// TwinCAT 3 PLC project MR1L0_MR2L0_PLC
// ProgramVersion: 3.1.4022.7
// libraries:
//   Tc2_ControllerToolbox, * (Beckhoff Automation GmbH)
//   Tc2_MC2, * (Beckhoff Automation GmbH)
//   Tc2_SerialCom, * (Beckhoff Automation GmbH)
//   Tc2_Standard, * (Beckhoff Automation GmbH)
//   Tc2_System, * (Beckhoff Automation GmbH)
//   Tc2_Utilities, * (Beckhoff Automation GmbH)
//   Tc3_Module, * (Beckhoff Automation GmbH)
//   VisuDialogs, * (System)
//   LCLS General,0.0.0,SLAC
//   lcls-twincat-motion,1.1.0,SLAC
//   lcls-twincat-optics,0.0.0,SLAC
// project tree:
//   / GlobalTextList.TcGTLO, PiezoDriver.TcTTO (not stored), PlcTask.TcTTO, SerialIO.TcTTO, Visualization Manager.TcVMO (not stored)
//   GVLs/ GVL_COM_Buffers.TcGVL, GVL_M1L0.TcGVL, GVL_M1L0_Constants.TcGVL, GVL_M2L0.TcGVL, GVL_M2L0_Constants.TcGVL, GVL_SerialIO.TcGVL
//   POUs/ Main.TcPOU
//   POUs/Serial Comm/ PiezoSerial.TcPOU, P_Serial_Com.TcPOU
// real-time tasks:
//   TASK PlcTask: cycle T#10ms, priority 20, ADS port 350
//   TASK PiezoDriver: cycle T#1ms, priority 3, ADS port 351
//   TASK SerialIO: cycle T#2ms, priority 1, ADS port 352
// motion (NC):
//   TASK NC-Task 1 SAF: cycle T#2ms, priority 4, ADS port 501
//   TASK NC-Task 1 SVB: cycle T#10ms, priority 8, ADS port 511
//   AXIS M1L0-Yup (id 1)
//     General: UnitName=um
//     Dynamic: Acceleration=200, Deceleration=200, DelayTime=0.008
//     Velo: Maximum=200
//     OtherSettings: AllowMotionCmdToSlave=true
//     encoder EncType=29
//       EncPara: ScaleFactorNumerator=0.001, MaxCount=#xffffffff, ReferenceSystem=1
//         SoftEndMinControl: Enable=true, Range=3133.7
//         SoftEndMaxControl: Enable=true, Range=27004.8
//         Inc: RefSoftSyncMask=#x0000ffff
//     drive DrvType=24
//       DrvPara: Inverse=true
//         Analog: VeloReferenz=488.28125, ScaleFactorActTorque=0.1
//         TimeComp: TaskDelayCycles=1
//     controller CtrType=2
//       CtrPara: PriorControlFactor=1
//         PosDiffControl: Range=100
//         PID: PosKp=50, PosExtKp=10, DeadBandPosition=0.3
//         Observer: BandWidth=20
//   AXIS M1L0-Ydwn (id 2)
//     General: UnitName=um
//     Dynamic: Acceleration=200, Deceleration=200, DelayTime=0.008
//     Velo: Maximum=200
//     OtherSettings: AllowMotionCmdToSlave=true
//     encoder EncType=29
//       EncPara: ScaleFactorNumerator=0.001, MaxCount=#xffffffff, ReferenceSystem=1
//         SoftEndMinControl: Enable=true, Range=2244.7
//         SoftEndMaxControl: Enable=true, Range=26310.2
//         Inc: RefSoftSyncMask=#x0000ffff
//     drive DrvType=24
//       DrvPara: Inverse=true
//         Analog: VeloReferenz=488.28125, ScaleFactorActTorque=0.1
//         TimeComp: TaskDelayCycles=1
//     controller CtrType=2
//       CtrPara: PriorControlFactor=1
//         PosDiffControl: Range=100
//         PID: PosKp=50, PosExtKp=10, DeadBandPosition=0.3
//         Observer: BandWidth=20
//   AXIS M1L0-Xup (id 3)
//     General: UnitName=um
//     Dynamic: Acceleration=2000, Deceleration=2000, DelayTime=0.008
//     Velo: Maximum=1000
//     OtherSettings: AllowMotionCmdToSlave=true
//     encoder EncType=29
//       EncPara: ScaleFactorNumerator=0.001, MaxCount=#xffffffff, ReferenceSystem=1
//         SoftEndMinControl: Enable=true, Range=24843
//         SoftEndMaxControl: Enable=true, Range=25581.9
//         Inc: RefSoftSyncMask=#x0000ffff
//     drive DrvType=24
//       Analog: VeloReferenz=1220.703125, ScaleFactorActTorque=0.1
//       TimeComp: TaskDelayCycles=1
//     controller CtrType=2
//       CtrPara: PriorControlFactor=1
//         PosDiffControl: Range=100
//         PID: PosKp=50, PosExtKp=50, DeadBandPosition=0.4
//         Observer: BandWidth=20
//   AXIS M1L0-Xdwn (id 4)
//     General: UnitName=um
//     Dynamic: Acceleration=2000, Deceleration=2000, DelayTime=0.008
//     Velo: Maximum=1000
//     OtherSettings: AllowMotionCmdToSlave=true
//     encoder EncType=29
//       EncPara: ScaleFactorNumerator=0.001, MaxCount=#xffffffff, ReferenceSystem=1
//         SoftEndMinControl: Range=24000
//         SoftEndMaxControl: Enable=true, Range=24518.2
//         Inc: RefSoftSyncMask=#x0000ffff
//     drive DrvType=24
//       DrvPara: Inverse=true
//         Analog: VeloReferenz=1220.703125, ScaleFactorActTorque=0.1
//         TimeComp: TaskDelayCycles=1
//     controller CtrType=2
//       CtrPara: PriorControlFactor=1
//         PosDiffControl: Range=100
//         PID: PosKp=50, PosExtKp=50, DeadBandPosition=0.4
//         Observer: BandWidth=20
//   AXIS M1L0-Pitch (id 5)
//     General: UnitName=urad
//     Dynamic: Acceleration=390, Deceleration=390, DelayTime=0.008
//     Velo: Maximum=150
//     OtherSettings: AllowMotionCmdToSlave=true
//     encoder EncType=29
//       EncPara: ScaleFactorNumerator=0.001949317739, MaxCount=#xffffffff, ReferenceSystem=1
//         SoftEndMinControl: Enable=true, Range=15600
//         SoftEndMaxControl: Enable=true, Range=21600
//         Inc: RefSoftSyncMask=#x0000ffff
//     drive DrvType=24
//       Analog: VeloReferenz=761.4522417, ScaleFactorActTorque=0.1
//       TimeComp: TaskDelayCycles=1
//     controller CtrType=2
//       CtrPara: PriorControlFactor=1
//         PosDiffControl: Range=150
//         PID: PosExtKp=1, DeadBandPosition=0.25
//         Observer: BandWidth=20
//   AXIS M1L0-Bender (id 6)
//     General: UnitName=um
//     Dynamic: Acceleration=150, Deceleration=150, DelayTime=0.008
//     Velo: Maximum=150
//     OtherSettings: AllowMotionCmdToSlave=true
//     encoder EncType=29
//       EncPara: ScaleFactorNumerator=0.001, MaxCount=#xffffffff, ReferenceSystem=1
//         SoftEndMinControl: Enable=true, Range=4268900
//         SoftEndMaxControl: Enable=true, Range=4278150
//         Inc: RefSoftSyncMask=#x0000ffff
//     drive DrvType=24
//       DrvPara: Inverse=true
//         Analog: VeloReferenz=195.3125, ScaleFactorActTorque=0.1
//         TimeComp: TaskDelayCycles=1
//     controller CtrType=2
//       CtrPara: PriorControlFactor=1
//         PID: PosKp=10, PosExtKp=0.001, PosExtVelo=0.9, DeadBandPosition=0.1
//         Observer: BandWidth=20
//   AXIS M2L0-Yup (id 7)
//     General: UnitName=um
//     Dynamic: Acceleration=200, Deceleration=200, DelayTime=0.008
//     Velo: Maximum=200
//     OtherSettings: AllowMotionCmdToSlave=true
//     encoder EncType=29
//       EncPara: ScaleFactorNumerator=0.001, MaxCount=#xffffffff, ReferenceSystem=1
//         SoftEndMinControl: Enable=true, Range=2500
//         SoftEndMaxControl: Enable=true, Range=18750
//         Inc: RefSoftSyncMask=#x0000ffff
//     drive DrvType=24
//       DrvPara: Inverse=true
//         Analog: VeloReferenz=488.28125, ScaleFactorActTorque=0.1
//         TimeComp: TaskDelayCycles=1
//     controller CtrType=2
//       CtrPara: PriorControlFactor=1
//         PosDiffControl: Range=100
//         PID: PosKp=20, PosExtKp=5, DeadBandPosition=0.4
//         Observer: BandWidth=20
//   AXIS M2L0-Ydwn (id 8)
//     General: UnitName=um
//     Dynamic: Acceleration=200, Deceleration=200, DelayTime=0.008
//     Velo: Maximum=200
//     OtherSettings: AllowMotionCmdToSlave=true
//     encoder EncType=29
//       EncPara: ScaleFactorNumerator=0.001, MaxCount=#xffffffff, ReferenceSystem=1
//         SoftEndMinControl: Enable=true, Range=5450
//         SoftEndMaxControl: Enable=true, Range=21800
//         Inc: RefSoftSyncMask=#x0000ffff
//     drive DrvType=24
//       DrvPara: Inverse=true
//         Analog: VeloReferenz=488.28125, ScaleFactorActTorque=0.1
//         TimeComp: TaskDelayCycles=1
//     controller CtrType=2
//       CtrPara: PriorControlFactor=1
//         PosDiffControl: Range=100
//         PID: PosKp=20, PosExtKp=5, DeadBandPosition=0.4
//         Observer: BandWidth=20
//   AXIS M2L0-Xup (id 9)
//     General: UnitName=um
//     Dynamic: Acceleration=2000, Deceleration=2000, DelayTime=0.008
//     Velo: Maximum=1000
//     OtherSettings: AllowMotionCmdToSlave=true
//     encoder EncType=29
//       EncPara: ScaleFactorNumerator=0.001, MaxCount=#xffffffff, ReferenceSystem=1
//         SoftEndMinControl: Enable=true, Range=24300
//         SoftEndMaxControl: Enable=true, Range=26200
//         Inc: RefSoftSyncMask=#x0000ffff
//     drive DrvType=24
//       Analog: VeloReferenz=1220.703125, ScaleFactorActTorque=0.1
//       TimeComp: TaskDelayCycles=1
//     controller CtrType=2
//       CtrPara: PriorControlFactor=1
//         PosDiffControl: Range=100
//         PID: PosKp=10, PosExtKp=1, DeadBandPosition=0.4
//         Observer: BandWidth=20
//   AXIS M2L0-Xdwn (id 10)
//     General: UnitName=um
//     Dynamic: Acceleration=2000, Deceleration=2000, DelayTime=0.008
//     Velo: Maximum=1000
//     OtherSettings: AllowMotionCmdToSlave=true
//     encoder EncType=29
//       EncPara: ScaleFactorNumerator=0.001, MaxCount=#xffffffff, ReferenceSystem=1
//         SoftEndMinControl: Range=23500
//         SoftEndMaxControl: Range=25700
//         Inc: RefSoftSyncMask=#x0000ffff
//     drive DrvType=24
//       DrvPara: Inverse=true
//         Analog: VeloReferenz=1220.703125, ScaleFactorActTorque=0.1
//         TimeComp: TaskDelayCycles=1
//     controller CtrType=2
//       CtrPara: PriorControlFactor=1
//         PosDiffControl: Range=100
//         PID: PosKp=10, PosExtKp=1, DeadBandPosition=0.4
//         Observer: BandWidth=20
//   AXIS M2L0-Pitch (id 11)
//     General: UnitName=urad
//     Dynamic: Acceleration=390, Deceleration=390
//     Velo: Maximum=150
//     OtherSettings: AllowMotionCmdToSlave=true
//     encoder EncType=29
//       EncPara: ScaleFactorNumerator=0.001949317739, MaxCount=#xffffffff, ReferenceSystem=1
//         SoftEndMinControl: Enable=true, Range=16200
//         SoftEndMaxControl: Enable=true, Range=20600
//         Inc: RefSoftSyncMask=#x0000ffff
//     drive DrvType=24
//       Analog: VeloReferenz=761.4522417, ScaleFactorActTorque=0.1
//       TimeComp: TaskDelayCycles=1
//     controller CtrType=2
//       CtrPara: PriorControlFactor=1
//         PosDiffControl: Range=150
//         PID: PosExtKp=1, DeadBandPosition=0.2
//         Observer: BandWidth=20
//   AXIS M2L0-Bender (id 12)
//     General: UnitName=um
//     Dynamic: Acceleration=150, Deceleration=150, DelayTime=0.008
//     Velo: Maximum=150
//     OtherSettings: AllowMotionCmdToSlave=true
//     encoder EncType=29
//       EncPara: ScaleFactorNumerator=0.001, MaxCount=#xffffffff, ReferenceSystem=1
//         SoftEndMinControl: Enable=true, Range=4268977
//         SoftEndMaxControl: Enable=true, Range=4279741
//         Inc: RefSoftSyncMask=#x0000ffff
//     drive DrvType=24
//       DrvPara: Inverse=true
//         Analog: VeloReferenz=195.3125, ScaleFactorActTorque=0.1
//         TimeComp: TaskDelayCycles=1
//     controller CtrType=2
//       CtrPara: PriorControlFactor=1
//         PID: PosKp=10, PosExtKp=0.001, PosExtVelo=0.9, DeadBandPosition=0.1
//         Observer: BandWidth=20
// I/O:
//   DEVICE Device 1 (EtherCAT), AmsNetId 172.21.88.30.2.1
//     Term 1 (EK1200)
// variable links:
//   (this object) <-> Device 1 (EtherCAT)/Term 1 (EK1200)/Term 5 (EK1122)/EK1100_M1L0/EL5042_M1L0_Yupdwn
//     Enc/Inputs/In/nComState @bit 1 <-> WcState/InputToggle
//     Enc/Inputs/In/nComState <-> WcState/WcState
//     Enc/Inputs/In/nDataIn1 <-> FB Inputs Channel 1/Position
//     Enc/Inputs/In/nDataIn1 <-> FB Inputs Channel 2/Position
//     Enc/Inputs/In/nState1 @bit 12 <-> FB Inputs Channel 1/Status/Diag
//     Enc/Inputs/In/nState1 @bit 12 <-> FB Inputs Channel 2/Status/Diag
//     Enc/Inputs/In/nState1 @bit 1 <-> FB Inputs Channel 1/Status/Error
//     Enc/Inputs/In/nState1 @bit 1 <-> FB Inputs Channel 2/Status/Error
//     Enc/Inputs/In/nState1 @bit 14 <-> FB Inputs Channel 1/Status/Input cycle counter
//     Enc/Inputs/In/nState1 @bit 14 <-> FB Inputs Channel 2/Status/Input cycle counter
//     Enc/Inputs/In/nState1 @bit 2 <-> FB Inputs Channel 1/Status/Ready
//     Enc/Inputs/In/nState1 @bit 2 <-> FB Inputs Channel 2/Status/Ready
//     Enc/Inputs/In/nState1 @bit 13 <-> FB Inputs Channel 1/Status/TxPDO State
//     Enc/Inputs/In/nState1 @bit 13 <-> FB Inputs Channel 2/Status/TxPDO State
//     Enc/Inputs/In/nState1 <-> FB Inputs Channel 1/Status/Warning
//     Enc/Inputs/In/nState1 <-> FB Inputs Channel 2/Status/Warning
//   (this object) <-> Device 1 (EtherCAT)/Term 1 (EK1200)/Term 5 (EK1122)/EK1100_M1L0/EL7041-1000_M1L0_Yup
//     Drive/Inputs/In/nState1 @bit 3 <-> STM Status/Status/Error
//     Drive/Inputs/In/nState1 @bit 5 <-> STM Status/Status/Moving negative
//     Drive/Inputs/In/nState1 @bit 4 <-> STM Status/Status/Moving positive
//     Drive/Inputs/In/nState1 @bit 1 <-> STM Status/Status/Ready
//     Drive/Inputs/In/nState1 <-> STM Status/Status/Ready to enable
//     Drive/Inputs/In/nState1 @bit 6 <-> STM Status/Status/Torque reduced
//     Drive/Inputs/In/nState1 @bit 2 <-> STM Status/Status/Warning
//     Drive/Inputs/In/nState2 @bit 3 <-> STM Status/Status/Digital input 1
//     Drive/Inputs/In/nState2 @bit 4 <-> STM Status/Status/Digital input 2
//     Drive/Inputs/In/nState2 @bit 5 <-> STM Status/Status/Sync error
//     Drive/Inputs/In/nState2 @bit 7 <-> STM Status/Status/TxPDO Toggle
//     Drive/Inputs/In/nState4 @bit 1 <-> WcState/InputToggle
//     Drive/Inputs/In/nState4 <-> WcState/WcState
//     Drive/Outputs/Out/nCtrl1 <-> STM Control/Control/Enable
//     Drive/Outputs/Out/nCtrl1 @bit 2 <-> STM Control/Control/Reduce torque
//     Drive/Outputs/Out/nCtrl1 @bit 1 <-> STM Control/Control/Reset
//     Drive/Outputs/Out/nDataOut2[0] <-> STM Velocity/Velocity
//   (this object) <-> Device 1 (EtherCAT)/Term 1 (EK1200)/Term 5 (EK1122)/EK1100_M1L0/EL7041-1000_M1L0_Ydwn
//     Drive/Inputs/In/nState1 @bit 3 <-> STM Status/Status/Error
//     Drive/Inputs/In/nState1 @bit 5 <-> STM Status/Status/Moving negative
//     Drive/Inputs/In/nState1 @bit 4 <-> STM Status/Status/Moving positive
//     Drive/Inputs/In/nState1 @bit 1 <-> STM Status/Status/Ready
//     Drive/Inputs/In/nState1 <-> STM Status/Status/Ready to enable
//     Drive/Inputs/In/nState1 @bit 6 <-> STM Status/Status/Torque reduced
//     Drive/Inputs/In/nState1 @bit 2 <-> STM Status/Status/Warning
//     Drive/Inputs/In/nState2 @bit 3 <-> STM Status/Status/Digital input 1
//     Drive/Inputs/In/nState2 @bit 4 <-> STM Status/Status/Digital input 2
//     Drive/Inputs/In/nState2 @bit 5 <-> STM Status/Status/Sync error
//     Drive/Inputs/In/nState2 @bit 7 <-> STM Status/Status/TxPDO Toggle
//     Drive/Inputs/In/nState4 @bit 1 <-> WcState/InputToggle
//     Drive/Inputs/In/nState4 <-> WcState/WcState
//     Drive/Outputs/Out/nCtrl1 <-> STM Control/Control/Enable
//     Drive/Outputs/Out/nCtrl1 @bit 2 <-> STM Control/Control/Reduce torque
//     Drive/Outputs/Out/nCtrl1 @bit 1 <-> STM Control/Control/Reset
//     Drive/Outputs/Out/nDataOut2[0] <-> STM Velocity/Velocity
//   (this object) <-> Device 1 (EtherCAT)/Term 1 (EK1200)/Term 5 (EK1122)/EK1100_M1L0/EL5042_M1L0_Xupdwn
//     Enc/Inputs/In/nComState @bit 1 <-> WcState/InputToggle
//     Enc/Inputs/In/nComState <-> WcState/WcState
//     Enc/Inputs/In/nDataIn1 <-> FB Inputs Channel 1/Position
//     Enc/Inputs/In/nDataIn1 <-> FB Inputs Channel 2/Position
//     Enc/Inputs/In/nState1 @bit 12 <-> FB Inputs Channel 1/Status/Diag
//     Enc/Inputs/In/nState1 @bit 12 <-> FB Inputs Channel 2/Status/Diag
//     Enc/Inputs/In/nState1 @bit 1 <-> FB Inputs Channel 1/Status/Error
//     Enc/Inputs/In/nState1 @bit 1 <-> FB Inputs Channel 2/Status/Error
//     Enc/Inputs/In/nState1 @bit 14 <-> FB Inputs Channel 1/Status/Input cycle counter
//     Enc/Inputs/In/nState1 @bit 14 <-> FB Inputs Channel 2/Status/Input cycle counter
//     Enc/Inputs/In/nState1 @bit 2 <-> FB Inputs Channel 1/Status/Ready
//     Enc/Inputs/In/nState1 @bit 2 <-> FB Inputs Channel 2/Status/Ready
//     Enc/Inputs/In/nState1 @bit 13 <-> FB Inputs Channel 1/Status/TxPDO State
//     Enc/Inputs/In/nState1 @bit 13 <-> FB Inputs Channel 2/Status/TxPDO State
//     Enc/Inputs/In/nState1 <-> FB Inputs Channel 1/Status/Warning
//     Enc/Inputs/In/nState1 <-> FB Inputs Channel 2/Status/Warning
//   (this object) <-> Device 1 (EtherCAT)/Term 1 (EK1200)/Term 5 (EK1122)/EK1100_M1L0/EL7041-1000_M1L0_Xup
//     Drive/Inputs/In/nState1 @bit 3 <-> STM Status/Status/Error
//     Drive/Inputs/In/nState1 @bit 5 <-> STM Status/Status/Moving negative
//     Drive/Inputs/In/nState1 @bit 4 <-> STM Status/Status/Moving positive
//     Drive/Inputs/In/nState1 @bit 1 <-> STM Status/Status/Ready
//     Drive/Inputs/In/nState1 <-> STM Status/Status/Ready to enable
//     Drive/Inputs/In/nState1 @bit 6 <-> STM Status/Status/Torque reduced
//     Drive/Inputs/In/nState1 @bit 2 <-> STM Status/Status/Warning
//     Drive/Inputs/In/nState2 @bit 3 <-> STM Status/Status/Digital input 1
//     Drive/Inputs/In/nState2 @bit 4 <-> STM Status/Status/Digital input 2
//     Drive/Inputs/In/nState2 @bit 5 <-> STM Status/Status/Sync error
//     Drive/Inputs/In/nState2 @bit 7 <-> STM Status/Status/TxPDO Toggle
//     Drive/Inputs/In/nState4 @bit 1 <-> WcState/InputToggle
//     Drive/Inputs/In/nState4 <-> WcState/WcState
//     Drive/Outputs/Out/nCtrl1 <-> STM Control/Control/Enable
//     Drive/Outputs/Out/nCtrl1 @bit 2 <-> STM Control/Control/Reduce torque
//     Drive/Outputs/Out/nCtrl1 @bit 1 <-> STM Control/Control/Reset
//     Drive/Outputs/Out/nDataOut2[0] <-> STM Velocity/Velocity
//   (this object) <-> Device 1 (EtherCAT)/Term 1 (EK1200)/Term 5 (EK1122)/EK1100_M1L0/EL7041-1000_M1L0_Xdwn
//     Drive/Inputs/In/nState1 @bit 3 <-> STM Status/Status/Error
//     Drive/Inputs/In/nState1 @bit 5 <-> STM Status/Status/Moving negative
//     Drive/Inputs/In/nState1 @bit 4 <-> STM Status/Status/Moving positive
//     Drive/Inputs/In/nState1 @bit 1 <-> STM Status/Status/Ready
//     Drive/Inputs/In/nState1 <-> STM Status/Status/Ready to enable
//     Drive/Inputs/In/nState1 @bit 6 <-> STM Status/Status/Torque reduced
//     Drive/Inputs/In/nState1 @bit 2 <-> STM Status/Status/Warning
//     Drive/Inputs/In/nState2 @bit 3 <-> STM Status/Status/Digital input 1
//     Drive/Inputs/In/nState2 @bit 4 <-> STM Status/Status/Digital input 2
//     Drive/Inputs/In/nState2 @bit 5 <-> STM Status/Status/Sync error
//     Drive/Inputs/In/nState2 @bit 7 <-> STM Status/Status/TxPDO Toggle
//     Drive/Inputs/In/nState4 @bit 1 <-> WcState/InputToggle
//     Drive/Inputs/In/nState4 <-> WcState/WcState
//     Drive/Outputs/Out/nCtrl1 <-> STM Control/Control/Enable
//     Drive/Outputs/Out/nCtrl1 @bit 2 <-> STM Control/Control/Reduce torque
//     Drive/Outputs/Out/nCtrl1 @bit 1 <-> STM Control/Control/Reset
//     Drive/Outputs/Out/nDataOut2[0] <-> STM Velocity/Velocity
//   (this object) <-> Device 1 (EtherCAT)/Term 1 (EK1200)/Term 5 (EK1122)/EK1100_M1L0/EL5042_M1L0_PitchBender
//     Enc/Inputs/In/nComState @bit 1 <-> WcState/InputToggle
//     Enc/Inputs/In/nComState <-> WcState/WcState
//     Enc/Inputs/In/nDataIn1 <-> FB Inputs Channel 1/Position
//     Enc/Inputs/In/nDataIn1 <-> FB Inputs Channel 2/Position
//     Enc/Inputs/In/nState1 @bit 12 <-> FB Inputs Channel 1/Status/Diag
//     Enc/Inputs/In/nState1 @bit 12 <-> FB Inputs Channel 2/Status/Diag
//     Enc/Inputs/In/nState1 @bit 1 <-> FB Inputs Channel 1/Status/Error
//     Enc/Inputs/In/nState1 @bit 1 <-> FB Inputs Channel 2/Status/Error
//     Enc/Inputs/In/nState1 @bit 14 <-> FB Inputs Channel 1/Status/Input cycle counter
//     Enc/Inputs/In/nState1 @bit 14 <-> FB Inputs Channel 2/Status/Input cycle counter
//     Enc/Inputs/In/nState1 @bit 2 <-> FB Inputs Channel 1/Status/Ready
//     Enc/Inputs/In/nState1 @bit 2 <-> FB Inputs Channel 2/Status/Ready
//     Enc/Inputs/In/nState1 @bit 13 <-> FB Inputs Channel 1/Status/TxPDO State
//     Enc/Inputs/In/nState1 @bit 13 <-> FB Inputs Channel 2/Status/TxPDO State
//     Enc/Inputs/In/nState1 <-> FB Inputs Channel 1/Status/Warning
//     Enc/Inputs/In/nState1 <-> FB Inputs Channel 2/Status/Warning
//   (this object) <-> Device 1 (EtherCAT)/Term 1 (EK1200)/Term 5 (EK1122)/EK1100_M1L0/EL7041-1000_M1L0_PitchCoarse
//     Drive/Inputs/In/nState1 @bit 3 <-> STM Status/Status/Error
//     Drive/Inputs/In/nState1 @bit 5 <-> STM Status/Status/Moving negative
//     Drive/Inputs/In/nState1 @bit 4 <-> STM Status/Status/Moving positive
//     Drive/Inputs/In/nState1 @bit 1 <-> STM Status/Status/Ready
//     Drive/Inputs/In/nState1 <-> STM Status/Status/Ready to enable
//     Drive/Inputs/In/nState1 @bit 6 <-> STM Status/Status/Torque reduced
//     Drive/Inputs/In/nState1 @bit 2 <-> STM Status/Status/Warning
//     Drive/Inputs/In/nState2 @bit 3 <-> STM Status/Status/Digital input 1
//     Drive/Inputs/In/nState2 @bit 4 <-> STM Status/Status/Digital input 2
//     Drive/Inputs/In/nState2 @bit 5 <-> STM Status/Status/Sync error
//     Drive/Inputs/In/nState2 @bit 7 <-> STM Status/Status/TxPDO Toggle
//     Drive/Inputs/In/nState4 @bit 1 <-> WcState/InputToggle
//     Drive/Inputs/In/nState4 <-> WcState/WcState
//     Drive/Outputs/Out/nCtrl1 <-> STM Control/Control/Enable
//     Drive/Outputs/Out/nCtrl1 @bit 2 <-> STM Control/Control/Reduce torque
//     Drive/Outputs/Out/nCtrl1 @bit 1 <-> STM Control/Control/Reset
//     Drive/Outputs/Out/nDataOut2[0] <-> STM Velocity/Velocity
//   (this object) <-> Device 1 (EtherCAT)/Term 1 (EK1200)/Term 5 (EK1122)/EK1100_M1L0/EL7041-1000_M1L0_Bender
//     Drive/Inputs/In/nState1 @bit 3 <-> STM Status/Status/Error
//     Drive/Inputs/In/nState1 @bit 5 <-> STM Status/Status/Moving negative
//     Drive/Inputs/In/nState1 @bit 4 <-> STM Status/Status/Moving positive
//     Drive/Inputs/In/nState1 @bit 1 <-> STM Status/Status/Ready
//     Drive/Inputs/In/nState1 <-> STM Status/Status/Ready to enable
//     Drive/Inputs/In/nState1 @bit 6 <-> STM Status/Status/Torque reduced
//     Drive/Inputs/In/nState1 @bit 2 <-> STM Status/Status/Warning
//     Drive/Inputs/In/nState2 @bit 3 <-> STM Status/Status/Digital input 1
//     Drive/Inputs/In/nState2 @bit 4 <-> STM Status/Status/Digital input 2
//     Drive/Inputs/In/nState2 @bit 5 <-> STM Status/Status/Sync error
//     Drive/Inputs/In/nState2 @bit 7 <-> STM Status/Status/TxPDO Toggle
//     Drive/Inputs/In/nState4 @bit 1 <-> WcState/InputToggle
//     Drive/Inputs/In/nState4 <-> WcState/WcState
//     Drive/Outputs/Out/nCtrl1 <-> STM Control/Control/Enable
//     Drive/Outputs/Out/nCtrl1 @bit 2 <-> STM Control/Control/Reduce torque
//     Drive/Outputs/Out/nCtrl1 @bit 1 <-> STM Control/Control/Reset
//     Drive/Outputs/Out/nDataOut2[0] <-> STM Velocity/Velocity
//   (this object) <-> Device 1 (EtherCAT)/Term 1 (EK1200)/Term 5 (EK1122)/EK1100_M2L0/EL5042_M2L0_Yupdwn
//     Enc/Inputs/In/nComState @bit 1 <-> WcState/InputToggle
//     Enc/Inputs/In/nComState <-> WcState/WcState
//     Enc/Inputs/In/nDataIn1 <-> FB Inputs Channel 1/Position
//     Enc/Inputs/In/nDataIn1 <-> FB Inputs Channel 2/Position
//     Enc/Inputs/In/nState1 @bit 12 <-> FB Inputs Channel 1/Status/Diag
//     Enc/Inputs/In/nState1 @bit 12 <-> FB Inputs Channel 2/Status/Diag
//     Enc/Inputs/In/nState1 @bit 1 <-> FB Inputs Channel 1/Status/Error
//     Enc/Inputs/In/nState1 @bit 1 <-> FB Inputs Channel 2/Status/Error
//     Enc/Inputs/In/nState1 @bit 14 <-> FB Inputs Channel 1/Status/Input cycle counter
//     Enc/Inputs/In/nState1 @bit 14 <-> FB Inputs Channel 2/Status/Input cycle counter
//     Enc/Inputs/In/nState1 @bit 2 <-> FB Inputs Channel 1/Status/Ready
//     Enc/Inputs/In/nState1 @bit 2 <-> FB Inputs Channel 2/Status/Ready
//     Enc/Inputs/In/nState1 @bit 13 <-> FB Inputs Channel 1/Status/TxPDO State
//     Enc/Inputs/In/nState1 @bit 13 <-> FB Inputs Channel 2/Status/TxPDO State
//     Enc/Inputs/In/nState1 <-> FB Inputs Channel 1/Status/Warning
//     Enc/Inputs/In/nState1 <-> FB Inputs Channel 2/Status/Warning
//   (this object) <-> Device 1 (EtherCAT)/Term 1 (EK1200)/Term 5 (EK1122)/EK1100_M2L0/EL7041-1000_M2L0_Yup
//     Drive/Inputs/In/nState1 @bit 3 <-> STM Status/Status/Error
//     Drive/Inputs/In/nState1 @bit 5 <-> STM Status/Status/Moving negative
//     Drive/Inputs/In/nState1 @bit 4 <-> STM Status/Status/Moving positive
//     Drive/Inputs/In/nState1 @bit 1 <-> STM Status/Status/Ready
//     Drive/Inputs/In/nState1 <-> STM Status/Status/Ready to enable
//     Drive/Inputs/In/nState1 @bit 6 <-> STM Status/Status/Torque reduced
//     Drive/Inputs/In/nState1 @bit 2 <-> STM Status/Status/Warning
//     Drive/Inputs/In/nState2 @bit 3 <-> STM Status/Status/Digital input 1
//     Drive/Inputs/In/nState2 @bit 4 <-> STM Status/Status/Digital input 2
//     Drive/Inputs/In/nState2 @bit 5 <-> STM Status/Status/Sync error
//     Drive/Inputs/In/nState2 @bit 7 <-> STM Status/Status/TxPDO Toggle
//     Drive/Inputs/In/nState4 @bit 1 <-> WcState/InputToggle
//     Drive/Inputs/In/nState4 <-> WcState/WcState
//     Drive/Outputs/Out/nCtrl1 <-> STM Control/Control/Enable
//     Drive/Outputs/Out/nCtrl1 @bit 2 <-> STM Control/Control/Reduce torque
//     Drive/Outputs/Out/nCtrl1 @bit 1 <-> STM Control/Control/Reset
//     Drive/Outputs/Out/nDataOut2[0] <-> STM Velocity/Velocity
//   (this object) <-> Device 1 (EtherCAT)/Term 1 (EK1200)/Term 5 (EK1122)/EK1100_M2L0/EL7041-1000_M2L0_Ydwn
//     Drive/Inputs/In/nState1 @bit 3 <-> STM Status/Status/Error
//     Drive/Inputs/In/nState1 @bit 5 <-> STM Status/Status/Moving negative
//     Drive/Inputs/In/nState1 @bit 4 <-> STM Status/Status/Moving positive
//     Drive/Inputs/In/nState1 @bit 1 <-> STM Status/Status/Ready
//     Drive/Inputs/In/nState1 <-> STM Status/Status/Ready to enable
//     Drive/Inputs/In/nState1 @bit 6 <-> STM Status/Status/Torque reduced
//     Drive/Inputs/In/nState1 @bit 2 <-> STM Status/Status/Warning
//     Drive/Inputs/In/nState2 @bit 3 <-> STM Status/Status/Digital input 1
//     Drive/Inputs/In/nState2 @bit 4 <-> STM Status/Status/Digital input 2
//     Drive/Inputs/In/nState2 @bit 5 <-> STM Status/Status/Sync error
//     Drive/Inputs/In/nState2 @bit 7 <-> STM Status/Status/TxPDO Toggle
//     Drive/Inputs/In/nState4 @bit 1 <-> WcState/InputToggle
//     Drive/Inputs/In/nState4 <-> WcState/WcState
//     Drive/Outputs/Out/nCtrl1 <-> STM Control/Control/Enable
//     Drive/Outputs/Out/nCtrl1 @bit 2 <-> STM Control/Control/Reduce torque
//     Drive/Outputs/Out/nCtrl1 @bit 1 <-> STM Control/Control/Reset
//     Drive/Outputs/Out/nDataOut2[0] <-> STM Velocity/Velocity
//   (this object) <-> Device 1 (EtherCAT)/Term 1 (EK1200)/Term 5 (EK1122)/EK1100_M2L0/EL5042_M2L0_Xupdwn
//     Enc/Inputs/In/nComState @bit 1 <-> WcState/InputToggle
//     Enc/Inputs/In/nComState <-> WcState/WcState
//     Enc/Inputs/In/nDataIn1 <-> FB Inputs Channel 1/Position
//     Enc/Inputs/In/nDataIn1 <-> FB Inputs Channel 2/Position
//     Enc/Inputs/In/nState1 @bit 12 <-> FB Inputs Channel 1/Status/Diag
//     Enc/Inputs/In/nState1 @bit 12 <-> FB Inputs Channel 2/Status/Diag
//     Enc/Inputs/In/nState1 @bit 1 <-> FB Inputs Channel 1/Status/Error
//     Enc/Inputs/In/nState1 @bit 1 <-> FB Inputs Channel 2/Status/Error
//     Enc/Inputs/In/nState1 @bit 14 <-> FB Inputs Channel 1/Status/Input cycle counter
//     Enc/Inputs/In/nState1 @bit 14 <-> FB Inputs Channel 2/Status/Input cycle counter
//     Enc/Inputs/In/nState1 @bit 2 <-> FB Inputs Channel 1/Status/Ready
//     Enc/Inputs/In/nState1 @bit 2 <-> FB Inputs Channel 2/Status/Ready
//     Enc/Inputs/In/nState1 @bit 13 <-> FB Inputs Channel 1/Status/TxPDO State
//     Enc/Inputs/In/nState1 @bit 13 <-> FB Inputs Channel 2/Status/TxPDO State
//     Enc/Inputs/In/nState1 <-> FB Inputs Channel 1/Status/Warning
//     Enc/Inputs/In/nState1 <-> FB Inputs Channel 2/Status/Warning
//   (this object) <-> Device 1 (EtherCAT)/Term 1 (EK1200)/Term 5 (EK1122)/EK1100_M2L0/EL7041-1000_M2L0_Xup
//     Drive/Inputs/In/nState1 @bit 3 <-> STM Status/Status/Error
//     Drive/Inputs/In/nState1 @bit 5 <-> STM Status/Status/Moving negative
//     Drive/Inputs/In/nState1 @bit 4 <-> STM Status/Status/Moving positive
//     Drive/Inputs/In/nState1 @bit 1 <-> STM Status/Status/Ready
//     Drive/Inputs/In/nState1 <-> STM Status/Status/Ready to enable
//     Drive/Inputs/In/nState1 @bit 6 <-> STM Status/Status/Torque reduced
//     Drive/Inputs/In/nState1 @bit 2 <-> STM Status/Status/Warning
//     Drive/Inputs/In/nState2 @bit 3 <-> STM Status/Status/Digital input 1
//     Drive/Inputs/In/nState2 @bit 4 <-> STM Status/Status/Digital input 2
//     Drive/Inputs/In/nState2 @bit 5 <-> STM Status/Status/Sync error
//     Drive/Inputs/In/nState2 @bit 7 <-> STM Status/Status/TxPDO Toggle
//     Drive/Inputs/In/nState4 @bit 1 <-> WcState/InputToggle
//     Drive/Inputs/In/nState4 <-> WcState/WcState
//     Drive/Outputs/Out/nCtrl1 <-> STM Control/Control/Enable
//     Drive/Outputs/Out/nCtrl1 @bit 2 <-> STM Control/Control/Reduce torque
//     Drive/Outputs/Out/nCtrl1 @bit 1 <-> STM Control/Control/Reset
//     Drive/Outputs/Out/nDataOut2[0] <-> STM Velocity/Velocity
//   (this object) <-> Device 1 (EtherCAT)/Term 1 (EK1200)/Term 5 (EK1122)/EK1100_M2L0/EL7041-1000_M2L0_Xdwn
//     Drive/Inputs/In/nState1 @bit 3 <-> STM Status/Status/Error
//     Drive/Inputs/In/nState1 @bit 5 <-> STM Status/Status/Moving negative
//     Drive/Inputs/In/nState1 @bit 4 <-> STM Status/Status/Moving positive
//     Drive/Inputs/In/nState1 @bit 1 <-> STM Status/Status/Ready
//     Drive/Inputs/In/nState1 <-> STM Status/Status/Ready to enable
//     Drive/Inputs/In/nState1 @bit 6 <-> STM Status/Status/Torque reduced
//     Drive/Inputs/In/nState1 @bit 2 <-> STM Status/Status/Warning
//     Drive/Inputs/In/nState2 @bit 3 <-> STM Status/Status/Digital input 1
//     Drive/Inputs/In/nState2 @bit 4 <-> STM Status/Status/Digital input 2
//     Drive/Inputs/In/nState2 @bit 5 <-> STM Status/Status/Sync error
//     Drive/Inputs/In/nState2 @bit 7 <-> STM Status/Status/TxPDO Toggle
//     Drive/Inputs/In/nState4 @bit 1 <-> WcState/InputToggle
//     Drive/Inputs/In/nState4 <-> WcState/WcState
//     Drive/Outputs/Out/nCtrl1 <-> STM Control/Control/Enable
//     Drive/Outputs/Out/nCtrl1 @bit 2 <-> STM Control/Control/Reduce torque
//     Drive/Outputs/Out/nCtrl1 @bit 1 <-> STM Control/Control/Reset
//     Drive/Outputs/Out/nDataOut2[0] <-> STM Velocity/Velocity
//   (this object) <-> Device 1 (EtherCAT)/Term 1 (EK1200)/Term 5 (EK1122)/EK1100_M2L0/EL5042_M2L0_PitchBender
//     Enc/Inputs/In/nComState @bit 1 <-> WcState/InputToggle
//     Enc/Inputs/In/nComState <-> WcState/WcState
//     Enc/Inputs/In/nDataIn1 <-> FB Inputs Channel 1/Position
//     Enc/Inputs/In/nDataIn1 <-> FB Inputs Channel 2/Position
//     Enc/Inputs/In/nState1 @bit 12 <-> FB Inputs Channel 1/Status/Diag
//     Enc/Inputs/In/nState1 @bit 12 <-> FB Inputs Channel 2/Status/Diag
//     Enc/Inputs/In/nState1 @bit 1 <-> FB Inputs Channel 1/Status/Error
//     Enc/Inputs/In/nState1 @bit 1 <-> FB Inputs Channel 2/Status/Error
//     Enc/Inputs/In/nState1 @bit 14 <-> FB Inputs Channel 1/Status/Input cycle counter
//     Enc/Inputs/In/nState1 @bit 14 <-> FB Inputs Channel 2/Status/Input cycle counter
//     Enc/Inputs/In/nState1 @bit 2 <-> FB Inputs Channel 1/Status/Ready
//     Enc/Inputs/In/nState1 @bit 2 <-> FB Inputs Channel 2/Status/Ready
//     Enc/Inputs/In/nState1 @bit 13 <-> FB Inputs Channel 1/Status/TxPDO State
//     Enc/Inputs/In/nState1 @bit 13 <-> FB Inputs Channel 2/Status/TxPDO State
//     Enc/Inputs/In/nState1 <-> FB Inputs Channel 1/Status/Warning
//     Enc/Inputs/In/nState1 <-> FB Inputs Channel 2/Status/Warning
//   (this object) <-> Device 1 (EtherCAT)/Term 1 (EK1200)/Term 5 (EK1122)/EK1100_M2L0/EL7041-1000_M2L0_PitchCoarse
//     Drive/Inputs/In/nState1 @bit 3 <-> STM Status/Status/Error
//     Drive/Inputs/In/nState1 @bit 5 <-> STM Status/Status/Moving negative
//     Drive/Inputs/In/nState1 @bit 4 <-> STM Status/Status/Moving positive
//     Drive/Inputs/In/nState1 @bit 1 <-> STM Status/Status/Ready
//     Drive/Inputs/In/nState1 <-> STM Status/Status/Ready to enable
//     Drive/Inputs/In/nState1 @bit 6 <-> STM Status/Status/Torque reduced
//     Drive/Inputs/In/nState1 @bit 2 <-> STM Status/Status/Warning
//     Drive/Inputs/In/nState2 @bit 3 <-> STM Status/Status/Digital input 1
//     Drive/Inputs/In/nState2 @bit 4 <-> STM Status/Status/Digital input 2
//     Drive/Inputs/In/nState2 @bit 5 <-> STM Status/Status/Sync error
//     Drive/Inputs/In/nState2 @bit 7 <-> STM Status/Status/TxPDO Toggle
//     Drive/Inputs/In/nState4 @bit 1 <-> WcState/InputToggle
//     Drive/Inputs/In/nState4 <-> WcState/WcState
//     Drive/Outputs/Out/nCtrl1 <-> STM Control/Control/Enable
//     Drive/Outputs/Out/nCtrl1 @bit 2 <-> STM Control/Control/Reduce torque
//     Drive/Outputs/Out/nCtrl1 @bit 1 <-> STM Control/Control/Reset
//     Drive/Outputs/Out/nDataOut2[0] <-> STM Velocity/Velocity
//   (this object) <-> Device 1 (EtherCAT)/Term 1 (EK1200)/Term 5 (EK1122)/EK1100_M2L0/EL7041-1000_M2L0_Bender
//     Drive/Inputs/In/nState1 @bit 3 <-> STM Status/Status/Error
//     Drive/Inputs/In/nState1 @bit 5 <-> STM Status/Status/Moving negative
//     Drive/Inputs/In/nState1 @bit 4 <-> STM Status/Status/Moving positive
//     Drive/Inputs/In/nState1 @bit 1 <-> STM Status/Status/Ready
//     Drive/Inputs/In/nState1 <-> STM Status/Status/Ready to enable
//     Drive/Inputs/In/nState1 @bit 6 <-> STM Status/Status/Torque reduced
//     Drive/Inputs/In/nState1 @bit 2 <-> STM Status/Status/Warning
//     Drive/Inputs/In/nState2 @bit 3 <-> STM Status/Status/Digital input 1
//     Drive/Inputs/In/nState2 @bit 4 <-> STM Status/Status/Digital input 2
//     Drive/Inputs/In/nState2 @bit 5 <-> STM Status/Status/Sync error
//     Drive/Inputs/In/nState2 @bit 7 <-> STM Status/Status/TxPDO Toggle
//     Drive/Inputs/In/nState4 @bit 1 <-> WcState/InputToggle
//     Drive/Inputs/In/nState4 <-> WcState/WcState
//     Drive/Outputs/Out/nCtrl1 <-> STM Control/Control/Enable
//     Drive/Outputs/Out/nCtrl1 @bit 2 <-> STM Control/Control/Reduce torque
//     Drive/Outputs/Out/nCtrl1 @bit 1 <-> STM Control/Control/Reset
//     Drive/Outputs/Out/nDataOut2[0] <-> STM Velocity/Velocity
//   MR1L0_MR2L0_PLC Instance <-> Device 1 (EtherCAT)
//     PlcTask Inputs/Main.fbECATDiag.arrEcMasterNetId <-> InfoData/AmsNetId
//     PlcTask Inputs/Main.fbECATDiag.nEcMasterDevState <-> Inputs/DevState
//     PlcTask Inputs/Main.fbECATDiag.nEcMasterDeviceId <-> InfoData/DevId
//     PlcTask Inputs/Main.fbECATDiag.nEcMasterSlaveCount <-> Inputs/SlaveCount
//     PlcTask Inputs/Main.fbECATDiag.nEcMasterSlaveCountCfg <-> InfoData/CfgSlaveCount
//     PlcTask Inputs/Main.fbECATDiag.wFrmXWcState <-> Inputs/Frm1WcState
//   MR1L0_MR2L0_PLC Instance <-> Device 1 (EtherCAT)/Term 1 (EK1200)/Term 5 (EK1122)/EK1100_M1L0/EL1004_M1L0_STO
//     PlcTask Inputs/Main.M1L0.fbRunHOMS.bSTOEnable1 <-> Channel 1/Input
//     PlcTask Inputs/Main.M1L0.fbRunHOMS.bSTOEnable2 <-> Channel 2/Input
//   MR1L0_MR2L0_PLC Instance <-> Device 1 (EtherCAT)/Term 1 (EK1200)/Term 5 (EK1122)/EK1100_M1L0/EL5042_M1L0_PitchBender
//     PlcTask Inputs/GVL_M1L0.M1L0_Pitch.diEncCnt <-> FB Inputs Channel 1/Position
//   MR1L0_MR2L0_PLC Instance <-> Device 1 (EtherCAT)/Term 1 (EK1200)/Term 5 (EK1122)/EK1100_M1L0/EL5042_M1L0_Xupdwn
//     PlcTask Inputs/Main.M1L0.fbRunHOMS.stXdwnEnc/Count <-> FB Inputs Channel 2/Position
//     PlcTask Inputs/Main.M1L0.fbRunHOMS.stXupEnc/Count <-> FB Inputs Channel 1/Position
//   MR1L0_MR2L0_PLC Instance <-> Device 1 (EtherCAT)/Term 1 (EK1200)/Term 5 (EK1122)/EK1100_M1L0/EL5042_M1L0_Yupdwn
//     PlcTask Inputs/Main.M1L0.fbRunHOMS.stYdwnEnc/Count <-> FB Inputs Channel 2/Position
//     PlcTask Inputs/Main.M1L0.fbRunHOMS.stYupEnc/Count <-> FB Inputs Channel 1/Position
//   MR1L0_MR2L0_PLC Instance <-> Device 1 (EtherCAT)/Term 1 (EK1200)/Term 5 (EK1122)/EK1100_M1L0/EL6001_M1L0_PitchFine
//     SerialIO Inputs/GVL_SerialIO.Serial_stComIn_M1L0/D[{0..21}] <-> COM Inputs/Data In {0..21}  (22 links)
//     SerialIO Inputs/GVL_SerialIO.Serial_stComIn_M1L0/Status <-> COM Inputs/Status
//     SerialIO Outputs/GVL_SerialIO.Serial_stComOut_M1L0/Ctrl <-> COM Outputs/Ctrl
//     SerialIO Outputs/GVL_SerialIO.Serial_stComOut_M1L0/D[{0..21}] <-> COM Outputs/Data Out {0..21}  (22 links)
//   MR1L0_MR2L0_PLC Instance <-> Device 1 (EtherCAT)/Term 1 (EK1200)/Term 5 (EK1122)/EK1100_M1L0/EL7041-1000_M1L0_Bender
//     PlcTask Inputs/Main.M6.bLimitBackwardEnable <-> STM Status/Status/Digital input 2
//     PlcTask Inputs/Main.M6.bLimitForwardEnable <-> STM Status/Status/Digital input 1
//   MR1L0_MR2L0_PLC Instance <-> Device 1 (EtherCAT)/Term 1 (EK1200)/Term 5 (EK1122)/EK1100_M1L0/EL7041-1000_M1L0_PitchCoarse
//     PlcTask Inputs/Main.M5.bLimitBackwardEnable <-> STM Status/Status/Digital input 2
//     PlcTask Inputs/Main.M5.bLimitForwardEnable <-> STM Status/Status/Digital input 1
//   MR1L0_MR2L0_PLC Instance <-> Device 1 (EtherCAT)/Term 1 (EK1200)/Term 5 (EK1122)/EK1100_M1L0/EL7041-1000_M1L0_Xdwn
//     PlcTask Inputs/Main.M4.bLimitBackwardEnable <-> STM Status/Status/Digital input 2
//     PlcTask Inputs/Main.M4.bLimitForwardEnable <-> STM Status/Status/Digital input 1
//   MR1L0_MR2L0_PLC Instance <-> Device 1 (EtherCAT)/Term 1 (EK1200)/Term 5 (EK1122)/EK1100_M1L0/EL7041-1000_M1L0_Xup
//     PlcTask Inputs/Main.M3.bLimitBackwardEnable <-> STM Status/Status/Digital input 2
//     PlcTask Inputs/Main.M3.bLimitForwardEnable <-> STM Status/Status/Digital input 1
//   MR1L0_MR2L0_PLC Instance <-> Device 1 (EtherCAT)/Term 1 (EK1200)/Term 5 (EK1122)/EK1100_M1L0/EL7041-1000_M1L0_Ydwn
//     PlcTask Inputs/Main.M2.bLimitBackwardEnable <-> STM Status/Status/Digital input 2
//     PlcTask Inputs/Main.M2.bLimitForwardEnable <-> STM Status/Status/Digital input 1
//   MR1L0_MR2L0_PLC Instance <-> Device 1 (EtherCAT)/Term 1 (EK1200)/Term 5 (EK1122)/EK1100_M1L0/EL7041-1000_M1L0_Yup
//     PlcTask Inputs/Main.M1.bLimitBackwardEnable <-> STM Status/Status/Digital input 2
//     PlcTask Inputs/Main.M1.bLimitForwardEnable <-> STM Status/Status/Digital input 1
//   MR1L0_MR2L0_PLC Instance <-> Device 1 (EtherCAT)/Term 1 (EK1200)/Term 5 (EK1122)/EK1100_M2L0/EL1004_M2L0_STO
//     PlcTask Inputs/Main.M2L0.fbRunHOMS.bSTOEnable1 <-> Channel 1/Input
//     PlcTask Inputs/Main.M2L0.fbRunHOMS.bSTOEnable2 <-> Channel 2/Input
//   MR1L0_MR2L0_PLC Instance <-> Device 1 (EtherCAT)/Term 1 (EK1200)/Term 5 (EK1122)/EK1100_M2L0/EL5042_M2L0_PitchBender
//     PlcTask Inputs/GVL_M2L0.M2L0_Pitch.diEncCnt <-> FB Inputs Channel 1/Position
//   MR1L0_MR2L0_PLC Instance <-> Device 1 (EtherCAT)/Term 1 (EK1200)/Term 5 (EK1122)/EK1100_M2L0/EL5042_M2L0_Xupdwn
//     PlcTask Inputs/Main.M2L0.fbRunHOMS.stXdwnEnc/Count <-> FB Inputs Channel 2/Position
//     PlcTask Inputs/Main.M2L0.fbRunHOMS.stXupEnc/Count <-> FB Inputs Channel 1/Position
//   MR1L0_MR2L0_PLC Instance <-> Device 1 (EtherCAT)/Term 1 (EK1200)/Term 5 (EK1122)/EK1100_M2L0/EL5042_M2L0_Yupdwn
//     PlcTask Inputs/Main.M2L0.fbRunHOMS.stYdwnEnc/Count <-> FB Inputs Channel 2/Position
//     PlcTask Inputs/Main.M2L0.fbRunHOMS.stYupEnc/Count <-> FB Inputs Channel 1/Position
//   MR1L0_MR2L0_PLC Instance <-> Device 1 (EtherCAT)/Term 1 (EK1200)/Term 5 (EK1122)/EK1100_M2L0/EL6001_M2L0_PitchFine
//     SerialIO Inputs/GVL_SerialIO.Serial_stComIn_M2L0/D[{0..21}] <-> COM Inputs/Data In {0..21}  (22 links)
//     SerialIO Inputs/GVL_SerialIO.Serial_stComIn_M2L0/Status <-> COM Inputs/Status
//     SerialIO Outputs/GVL_SerialIO.Serial_stComOut_M2L0/Ctrl <-> COM Outputs/Ctrl
//     SerialIO Outputs/GVL_SerialIO.Serial_stComOut_M2L0/D[{0..21}] <-> COM Outputs/Data Out {0..21}  (22 links)
//   MR1L0_MR2L0_PLC Instance <-> Device 1 (EtherCAT)/Term 1 (EK1200)/Term 5 (EK1122)/EK1100_M2L0/EL7041-1000_M2L0_Bender
//     PlcTask Inputs/Main.M12.bLimitBackwardEnable <-> STM Status/Status/Digital input 2
//     PlcTask Inputs/Main.M12.bLimitForwardEnable <-> STM Status/Status/Digital input 1
//   MR1L0_MR2L0_PLC Instance <-> Device 1 (EtherCAT)/Term 1 (EK1200)/Term 5 (EK1122)/EK1100_M2L0/EL7041-1000_M2L0_PitchCoarse
//     PlcTask Inputs/Main.M11.bLimitBackwardEnable <-> STM Status/Status/Digital input 2
//     PlcTask Inputs/Main.M11.bLimitForwardEnable <-> STM Status/Status/Digital input 1
//   MR1L0_MR2L0_PLC Instance <-> Device 1 (EtherCAT)/Term 1 (EK1200)/Term 5 (EK1122)/EK1100_M2L0/EL7041-1000_M2L0_Xdwn
//     PlcTask Inputs/Main.M10.bLimitBackwardEnable <-> STM Status/Status/Digital input 2
//     PlcTask Inputs/Main.M10.bLimitForwardEnable <-> STM Status/Status/Digital input 1
//   MR1L0_MR2L0_PLC Instance <-> Device 1 (EtherCAT)/Term 1 (EK1200)/Term 5 (EK1122)/EK1100_M2L0/EL7041-1000_M2L0_Xup
//     PlcTask Inputs/Main.M9.bLimitBackwardEnable <-> STM Status/Status/Digital input 2
//     PlcTask Inputs/Main.M9.bLimitForwardEnable <-> STM Status/Status/Digital input 1
//   MR1L0_MR2L0_PLC Instance <-> Device 1 (EtherCAT)/Term 1 (EK1200)/Term 5 (EK1122)/EK1100_M2L0/EL7041-1000_M2L0_Ydwn
//     PlcTask Inputs/Main.M8.bLimitBackwardEnable <-> STM Status/Status/Digital input 2
//     PlcTask Inputs/Main.M8.bLimitForwardEnable <-> STM Status/Status/Digital input 1
//   MR1L0_MR2L0_PLC Instance <-> Device 1 (EtherCAT)/Term 1 (EK1200)/Term 5 (EK1122)/EK1100_M2L0/EL7041-1000_M2L0_Yup
//     PlcTask Inputs/Main.M7.bLimitBackwardEnable <-> STM Status/Status/Digital input 2
//     PlcTask Inputs/Main.M7.bLimitForwardEnable <-> STM Status/Status/Digital input 1
//   MR1L0_MR2L0_PLC Instance <-> NC-Task 1 SAF/Axes/M1L0-Bender
//     PlcTask Inputs/Main.M6.Axis.NcToPlc <-> Outputs/ToPlc
//     PlcTask Outputs/Main.M6.Axis.PlcToNc <-> Inputs/FromPlc
//   MR1L0_MR2L0_PLC Instance <-> NC-Task 1 SAF/Axes/M1L0-Pitch
//     PlcTask Inputs/Main.M5.Axis.NcToPlc <-> Outputs/ToPlc
//     PlcTask Outputs/Main.M5.Axis.PlcToNc <-> Inputs/FromPlc
//   MR1L0_MR2L0_PLC Instance <-> NC-Task 1 SAF/Axes/M1L0-Xdwn
//     PlcTask Inputs/Main.M4.Axis.NcToPlc <-> Outputs/ToPlc
//     PlcTask Outputs/Main.M4.Axis.PlcToNc <-> Inputs/FromPlc
//   MR1L0_MR2L0_PLC Instance <-> NC-Task 1 SAF/Axes/M1L0-Xup
//     PlcTask Inputs/Main.M3.Axis.NcToPlc <-> Outputs/ToPlc
//     PlcTask Outputs/Main.M3.Axis.PlcToNc <-> Inputs/FromPlc
//   MR1L0_MR2L0_PLC Instance <-> NC-Task 1 SAF/Axes/M1L0-Ydwn
//     PlcTask Inputs/Main.M2.Axis.NcToPlc <-> Outputs/ToPlc
//     PlcTask Outputs/Main.M2.Axis.PlcToNc <-> Inputs/FromPlc
//   MR1L0_MR2L0_PLC Instance <-> NC-Task 1 SAF/Axes/M1L0-Yup
//     PlcTask Inputs/Main.M1.Axis.NcToPlc <-> Outputs/ToPlc
//     PlcTask Outputs/Main.M1.Axis.PlcToNc <-> Inputs/FromPlc
//   MR1L0_MR2L0_PLC Instance <-> NC-Task 1 SAF/Axes/M2L0-Bender
//     PlcTask Inputs/Main.M12.Axis.NcToPlc <-> Outputs/ToPlc
//     PlcTask Outputs/Main.M12.Axis.PlcToNc <-> Inputs/FromPlc
//   MR1L0_MR2L0_PLC Instance <-> NC-Task 1 SAF/Axes/M2L0-Pitch
//     PlcTask Inputs/Main.M11.Axis.NcToPlc <-> Outputs/ToPlc
//     PlcTask Outputs/Main.M11.Axis.PlcToNc <-> Inputs/FromPlc
//   MR1L0_MR2L0_PLC Instance <-> NC-Task 1 SAF/Axes/M2L0-Xdwn
//     PlcTask Inputs/Main.M10.Axis.NcToPlc <-> Outputs/ToPlc
//     PlcTask Outputs/Main.M10.Axis.PlcToNc <-> Inputs/FromPlc
//   MR1L0_MR2L0_PLC Instance <-> NC-Task 1 SAF/Axes/M2L0-Xup
//     PlcTask Inputs/Main.M9.Axis.NcToPlc <-> Outputs/ToPlc
//     PlcTask Outputs/Main.M9.Axis.PlcToNc <-> Inputs/FromPlc
//   MR1L0_MR2L0_PLC Instance <-> NC-Task 1 SAF/Axes/M2L0-Ydwn
//     PlcTask Inputs/Main.M8.Axis.NcToPlc <-> Outputs/ToPlc
//     PlcTask Outputs/Main.M8.Axis.PlcToNc <-> Inputs/FromPlc
//   MR1L0_MR2L0_PLC Instance <-> NC-Task 1 SAF/Axes/M2L0-Yup
//     PlcTask Inputs/Main.M7.Axis.NcToPlc <-> Outputs/ToPlc
//     PlcTask Outputs/Main.M7.Axis.PlcToNc <-> Inputs/FromPlc

CONFIGURATION MR1L0_MR2L0_PLC
    RESOURCE PLC ON TwinCAT3
        TASK PlcTask(INTERVAL := T#10ms, PRIORITY := 20);
        TASK SerialIO(INTERVAL := T#2ms, PRIORITY := 1);
        PROGRAM Main WITH PlcTask : Main;
        PROGRAM P_Serial_Com WITH SerialIO : P_Serial_Com;
    END_RESOURCE
END_CONFIGURATION

// ---- GVLs/GVL_COM_Buffers.TcGVL
VAR_GLOBAL
	// M1L0
	Serial_RXBuffer_M1L0 : ComBuffer;
	Serial_TXBuffer_M1L0 : ComBuffer;

	// M2L0
	Serial_RXBuffer_M2L0 : ComBuffer;
	Serial_TXBuffer_M2L0 : ComBuffer;
END_VAR

// ---- GVLs/GVL_M1L0.TcGVL
{attribute 'qualified_only'}
VAR_GLOBAL
	// Pitch Mechanism:
	{attribute 'TcLinkTo' := '.diEncCnt:=TIIB[EL5042_M1L0_PitchBender]^FB Inputs Channel 1^Position'}
	M1L0_Pitch : HOMS_PitchMechanism := (ReqPosLimHi := 21500,
		                                 ReqPosLimLo := 15500,
		                                 diEncPosLimHi := 11029500,
		                                 diEncPosLimLo := 7951500);
END_VAR

// ---- GVLs/GVL_M1L0_Constants.TcGVL
{attribute 'qualified_only'}
VAR_GLOBAL CONSTANT
	// Encoder reference values in counts = nm
	// Enc Ref Vals from alignment 2020-3-13
	nYUP_ENC_REF : ULINT := 15417790;
	nYDWN_ENC_REF : ULINT := 14628620;
	nXUP_ENC_REF : ULINT := 25479550;
	nXDWN_ENC_REF : ULINT := 24312380;
END_VAR

// ---- GVLs/GVL_M2L0.TcGVL
{attribute 'qualified_only'}
VAR_GLOBAL
	// Pitch Mechanism
	{attribute 'TcLinkTo' := '.diEncCnt:=TIIB[EL5042_M2L0_PitchBender]^FB Inputs Channel 1^Position'}
	M2L0_Pitch : HOMS_PitchMechanism := (ReqPosLimHi := 20000,
		                                 ReqPosLimLo := 17000,
		                                 diEncPosLimHi := 10260000,
		                                 diEncPosLimLo := 8721000);
END_VAR

// ---- GVLs/GVL_M2L0_Constants.TcGVL
{attribute 'qualified_only'}
VAR_GLOBAL CONSTANT
	// Encoder reference values in counts = nm
	// Encoder reference values after alignment 3-13-20
	nYUP_ENC_REF : ULINT := 11805150;
	nYDWN_ENC_REF : ULINT := 14830760;
	nXUP_ENC_REF : ULINT := 25288760;
	nXDWN_ENC_REF : ULINT := 24194070;
END_VAR

// ---- GVLs/GVL_SerialIO.TcGVL
VAR_GLOBAL
	//Better have your inputs and outputs!
	// M1L0
	Serial_stComIn_M1L0   AT %I*	:	EL6inData22B (*KL6inData22B*);
	Serial_stComOut_M1L0  AT %Q*	:	EL6outData22B (*KL6outData22B*);

	// M2L0
	Serial_stComIn_M2L0   AT %I*	:	EL6inData22B (*KL6inData22B*);
	Serial_stComOut_M2L0  AT %Q*	:	EL6outData22B (*KL6outData22B*);
END_VAR

// ---- POUs/Main.TcPOU
PROGRAM Main
VAR
	// M1L0
	// Motors
	{attribute 'TcLinkTo' := '.bLimitForwardEnable:=TIIB[EL7041-1000_M1L0_Yup]^STM Status^Status^Digital input 1;
                              .bLimitBackwardEnable:=TIIB[EL7041-1000_M1L0_Yup]^STM Status^Status^Digital input 2'}
	{attribute 'pytmc' := '
		pv: MR1L0:MMS:YUP
	'}
	M1 : DUT_MotionStage := (fVelocity:=200.0, nEnableMode:=ENUM_StageEnableMode.ALWAYS); // M1L0 Yup
	fbMotionStage_m1 : FB_MotionStage;

	{attribute 'TcLinkTo' := '.bLimitForwardEnable:=TIIB[EL7041-1000_M1L0_Ydwn]^STM Status^Status^Digital input 1;
                              .bLimitBackwardEnable:=TIIB[EL7041-1000_M1L0_Ydwn]^STM Status^Status^Digital input 2'}
	{attribute 'pytmc' := '
		pv: MR1L0:MMS:YDWN
	'}
	M2 : DUT_MotionStage := (fVelocity:=200.0, nEnableMode:=ENUM_StageEnableMode.ALWAYS); // M1L0 Ydwn
	fbMotionStage_m2 : FB_MotionStage;

	{attribute 'TcLinkTo' := '.bLimitForwardEnable:=TIIB[EL7041-1000_M1L0_Xup]^STM Status^Status^Digital input 1;
                              .bLimitBackwardEnable:=TIIB[EL7041-1000_M1L0_Xup]^STM Status^Status^Digital input 2'}
	{attribute 'pytmc' := '
		pv: MR1L0:MMS:XUP
	'}
	M3 : DUT_MotionStage := (fVelocity:=1000.0, nEnableMode:=ENUM_StageEnableMode.ALWAYS); // M1L0 Xup
	fbMotionStage_m3 : FB_MotionStage;

	{attribute 'TcLinkTo' := '.bLimitForwardEnable:=TIIB[EL7041-1000_M1L0_Xdwn]^STM Status^Status^Digital input 1;
                              .bLimitBackwardEnable:=TIIB[EL7041-1000_M1L0_Xdwn]^STM Status^Status^Digital input 2'}
	{attribute 'pytmc' := '
		pv: MR1L0:MMS:XDWN
	'}
	M4 : DUT_MotionStage := (fVelocity:=1000.0, nEnableMode:=ENUM_StageEnableMode.ALWAYS); // M1L0 Xdwn
	fbMotionStage_m4 : FB_MotionStage;

	{attribute 'TcLinkTo' := '.bLimitForwardEnable:=TIIB[EL7041-1000_M1L0_PitchCoarse]^STM Status^Status^Digital input 1;
                              .bLimitBackwardEnable:=TIIB[EL7041-1000_M1L0_PitchCoarse]^STM Status^Status^Digital input 2'}
	{attribute 'pytmc' := '
		pv: MR1L0:MMS:PITCH
	'}
	M5 : DUT_MotionStage := (fVelocity:=150.0); // M1L0 Pitch Stepper

	{attribute 'TcLinkTo' := '.bLimitForwardEnable:=TIIB[EL7041-1000_M1L0_Bender]^STM Status^Status^Digital input 1;
                              .bLimitBackwardEnable:=TIIB[EL7041-1000_M1L0_Bender]^STM Status^Status^Digital input 2'}
	{attribute 'pytmc' := '
		pv: MR1L0:MMS:BENDER
	'}
	M6 : DUT_MotionStage := (fVelocity:=150.0, nEnableMode:=ENUM_StageEnableMode.ALWAYS); // M1L0 Bender
	fbMotionStage_m6 : FB_MotionStage;

	{attribute 'TcLinkTo' := '.fbRunHOMS.bSTOEnable1:=TIIB[EL1004_M1L0_STO]^Channel 1^Input;
                              .fbRunHOMS.bSTOEnable2:=TIIB[EL1004_M1L0_STO]^Channel 2^Input;
	                          .fbRunHOMS.stYupEnc.Count:=TIIB[EL5042_M1L0_Yupdwn]^FB Inputs Channel 1^Position;
	                          .fbRunHOMS.stYdwnEnc.Count:=TIIB[EL5042_M1L0_Yupdwn]^FB Inputs Channel 2^Position;
	                          .fbRunHOMS.stXupEnc.Count:=TIIB[EL5042_M1L0_Xupdwn]^FB Inputs Channel 1^Position;
	                          .fbRunHOMS.stXdwnEnc.Count:=TIIB[EL5042_M1L0_Xupdwn]^FB Inputs Channel 2^Position'}
	{attribute 'pytmc' := '
		pv: MR1L0
	'}
	M1L0 : DUT_HOMS;

	// Encoder Arrays/RMS Watch:
	{attribute 'pytmc' := '
		pv: MR1L0:ENC:Y
	'}
	fbYRMSErrorM1L0 : FB_RMSWatch;
	fMaxYRMSErrorM1L0 : LREAL;
	fMinYRMSErrorM1L0 : LREAL;

	{attribute 'pytmc' := '
		pv: MR1L0:ENC:X
	'}
	fbXRMSErrorM1L0 : FB_RMSWatch;
	fMaxXRMSErrorM1L0 : LREAL;
	fMinXRMSErrorM1L0 : LREAL;

	{attribute 'pytmc' := '
		pv: MR1L0:ENC:PITCH
	'}
	fbPitchRMSErrorM1L0 : FB_RMSWatch;
	fMaxPitchRMSErrorM1L0 : LREAL;
	fMinPitchRMSErrorM1L0 : LREAL;

	{attribute 'pytmc' := '
		pv: MR1L0:ENC:BENDER
	'}
	fbBenderRMSErrorM1L0 : FB_RMSWatch;
	fMaxBenderRMSErrorM1L0 : LREAL;
	fMinBenderRMSErrorM1L0 : LREAL;

	// Pitch Control
	fbM1L0PitchControl : FB_PitchControl;
	bM1L0PitchDone : BOOL;
	bM1L0PitchBusy : BOOL;

	// Bender Control
	fbBenderM1L0 : FB_Bender;


	// M2L0
	// Motors
	{attribute 'TcLinkTo' := '.bLimitForwardEnable:=TIIB[EL7041-1000_M2L0_Yup]^STM Status^Status^Digital input 1;
                              .bLimitBackwardEnable:=TIIB[EL7041-1000_M2L0_Yup]^STM Status^Status^Digital input 2'}
	{attribute 'pytmc' := '
		pv: MR2L0:MMS:YUP
	'}
	M7 : DUT_MotionStage := (fVelocity:=200.0, nEnableMode:=ENUM_StageEnableMode.ALWAYS); // M2L0 Yup
	fbMotionStage_m7 : FB_MotionStage;

	{attribute 'TcLinkTo' := '.bLimitForwardEnable:=TIIB[EL7041-1000_M2L0_Ydwn]^STM Status^Status^Digital input 1;
                              .bLimitBackwardEnable:=TIIB[EL7041-1000_M2L0_Ydwn]^STM Status^Status^Digital input 2'}
	{attribute 'pytmc' := '
		pv: MR2L0:MMS:YDWN
	'}
	M8 : DUT_MotionStage := (fVelocity:=200.0, nEnableMode:=ENUM_StageEnableMode.ALWAYS); // M2L0 Ydwn
	fbMotionStage_m8 : FB_MotionStage;

	{attribute 'TcLinkTo' := '.bLimitForwardEnable:=TIIB[EL7041-1000_M2L0_Xup]^STM Status^Status^Digital input 1;
                              .bLimitBackwardEnable:=TIIB[EL7041-1000_M2L0_Xup]^STM Status^Status^Digital input 2'}
	{attribute 'pytmc' := '
		pv: MR2L0:MMS:XUP
	'}
	M9 : DUT_MotionStage := (fVelocity:=1000.0, nEnableMode:=ENUM_StageEnableMode.ALWAYS); // M2L0 Xup
	fbMotionStage_m9 : FB_MotionStage;

	{attribute 'TcLinkTo' := '.bLimitForwardEnable:=TIIB[EL7041-1000_M2L0_Xdwn]^STM Status^Status^Digital input 1;
                              .bLimitBackwardEnable:=TIIB[EL7041-1000_M2L0_Xdwn]^STM Status^Status^Digital input 2'}
	{attribute 'pytmc' := '
		pv: MR2L0:MMS:XDWN
	'}
	M10 : DUT_MotionStage := (fVelocity:=1000.0, nEnableMode:=ENUM_StageEnableMode.ALWAYS); // M2L0 Xdwn
	fbMotionStage_m10 : FB_MotionStage;
	
	{attribute 'TcLinkTo' := '.bLimitForwardEnable:=TIIB[EL7041-1000_M2L0_PitchCoarse]^STM Status^Status^Digital input 1;
                              .bLimitBackwardEnable:=TIIB[EL7041-1000_M2L0_PitchCoarse]^STM Status^Status^Digital input 2'}
	{attribute 'pytmc' := '
		pv: MR2L0:MMS:PITCH
	'}
	M11 : DUT_MotionStage := (fVelocity:=150.0); // M2L0 Pitch Stepper

	{attribute 'TcLinkTo' := '.bLimitForwardEnable:=TIIB[EL7041-1000_M2L0_Bender]^STM Status^Status^Digital input 1;
                              .bLimitBackwardEnable:=TIIB[EL7041-1000_M2L0_Bender]^STM Status^Status^Digital input 2'}
	{attribute 'pytmc' := '
		pv: MR2L0:MMS:BENDER
	'}
	M12 : DUT_MotionStage := (fVelocity:=150.0, nEnableMode:=ENUM_StageEnableMode.ALWAYS); // M2L0 Bender
	fbMotionStage_m12 : FB_MotionStage;

	{attribute 'TcLinkTo' := '.fbRunHOMS.bSTOEnable1:=TIIB[EL1004_M2L0_STO]^Channel 1^Input;
	                          .fbRunHOMS.bSTOEnable2:=TIIB[EL1004_M2L0_STO]^Channel 2^Input;
	                          .fbRunHOMS.stYupEnc.Count:=TIIB[EL5042_M2L0_Yupdwn]^FB Inputs Channel 1^Position;
	                          .fbRunHOMS.stYdwnEnc.Count:=TIIB[EL5042_M2L0_Yupdwn]^FB Inputs Channel 2^Position;
	                          .fbRunHOMS.stXupEnc.Count:=TIIB[EL5042_M2L0_Xupdwn]^FB Inputs Channel 1^Position;
	                          .fbRunHOMS.stXdwnEnc.Count:=TIIB[EL5042_M2L0_Xupdwn]^FB Inputs Channel 2^Position'}
	{attribute 'pytmc' := '
		pv: MR2L0
	'}
	M2L0 : DUT_HOMS;

	// Encoder Arrays/RMS Watch:
	{attribute 'pytmc' := '
		pv: MR2L0:ENC:Y
	'}
	fbYRMSErrorM2L0 : FB_RMSWatch;
	fMaxYRMSErrorM2L0 : LREAL;
	fMinYRMSErrorM2L0 : LREAL;

	{attribute 'pytmc' := '
		pv: MR2L0:ENC:X
	'}
	fbXRMSErrorM2L0 : FB_RMSWatch;
	fMaxXRMSErrorM2L0 : LREAL;
	fMinXRMSErrorM2L0 : LREAL;

	{attribute 'pytmc' := '
		pv: MR2L0:ENC:PITCH
	'}
	fbPitchRMSErrorM2L0 : FB_RMSWatch;
	fMaxPitchRMSErrorM2L0 : LREAL;
	fMinPitchRMSErrorM2L0 : LREAL;

	{attribute 'pytmc' := '
		pv: MR2L0:ENC:BENDER
	'}
	fbBenderRMSErrorM2L0 : FB_RMSWatch;
	fMaxBenderRMSErrorM2L0 : LREAL;
	fMinBenderRMSErrorM2L0 : LREAL;

	// Pitch Control
	fbM2L0PitchControl : FB_PitchControl;
	bM2L0PitchDone : BOOL;
	bM2L0PitchBusy : BOOL;

	// Bender Control
	fbBenderM2L0 : FB_Bender;
	
	// Logging
	fbLogHandler : FB_LogHandler;
	fbECATDiag : FB_EcatDiagWrapper;
END_VAR

// M1L0
M1L0.fbRunHOMS(stYup:=M1,
               stYdwn:=M2,
               stXup:=M3,
               stXdwn:=M4,
               stPitch:=M5,
	           nYupEncRef:=GVL_M1L0_Constants.nYUP_ENC_REF,
               nYdwnEncRef:=GVL_M1L0_Constants.nYDWN_ENC_REF,
               nXupEncRef:=GVL_M1L0_Constants.nXUP_ENC_REF,
               nXdwnEncRef:=GVL_M1L0_Constants.nXDWN_ENC_REF,
			   bExecuteCoupleY:=M1L0.bExecuteCoupleY,
               bExecuteCoupleX:=M1L0.bExecuteCoupleX,
			   bExecuteDecoupleY:=M1L0.bExecuteDecoupleY,
               bExecuteDecoupleX:=M1L0.bExecuteDecoupleX,
               bGantryAlreadyCoupledY=>M1L0.bGantryAlreadyCoupledY,
               bGantryAlreadyCoupledX=>M1L0.bGantryAlreadyCoupledX,
               nCurrGantryY=>M1L0.nCurrGantryY,
               nCurrGantryX=>M1L0.nCurrGantryX);
fbBenderM1L0(stBender:=M6,
	         bSTOEnable1:=M1L0.fbRunHOMS.bSTOEnable1,
		     bSTOEnable2:=M1L0.fbRunHOMS.bSTOEnable2);

// Convert nCurrGantry to um (smaller number) to read out in epics
M1L0.fCurrGantryY_um := LINT_TO_REAL(M1L0.nCurrGantryY) / 1000.0;
M1L0.fCurrGantryX_um := LINT_TO_REAL(M1L0.nCurrGantryX) / 1000.0;

// FB_MotionStage's for non-piezo axes
fbMotionStage_m1(stMotionStage:=M1);
fbMotionStage_m2(stMotionStage:=M2);
fbMotionStage_m3(stMotionStage:=M3);
fbMotionStage_m4(stMotionStage:=M4);
fbMotionStage_m6(stMotionStage:=M6);

// Calculate Pitch RMS Error:
fbYRMSErrorM1L0(stMotionStage:=M1,
	            fMaxRMSError=>fMaxYRMSErrorM1L0,
				fMinRMSError=>fMinYRMSErrorM1L0);

fbXRMSErrorM1L0(stMotionStage:=M3,
	            fMaxRMSError=>fMaxXRMSErrorM1L0,
				fMinRMSError=>fMinXRMSErrorM1L0);

fbPitchRMSErrorM1L0(stMotionStage:=M5,
	                fMaxRMSError=>fMaxPitchRMSErrorM1L0,
					fMinRMSError=>fMinPitchRMSErrorM1L0);

fbBenderRMSErrorM1L0(stMotionStage:=M6,
	                 fMaxRMSError=>fMaxBenderRMSErrorM1L0,
					 fMinRMSError=>fMinBenderRMSErrorM1L0);
// Pitch Control
fbM1L0PitchControl(Pitch:=GVL_M1L0.M1L0_Pitch,
				   Stepper:=M5,
				   lrCurrentSetpoint:=M5.fPosition,
                   q_bDone=>bM1L0PitchDone,
                   q_bBusy=>bM1L0PitchBusy);
// When STO hit, need to reset SP
IF NOT M5.bHardwareEnable THEN
	M5.fPosition := M5.stAxisStatus.fActPosition;
END_IF

// M2L0
M2L0.fbRunHOMS(stYup:=M7,
               stYdwn:=M8,
               stXup:=M9,
               stXdwn:=M10,
			   stPitch:=M11,
	           nYupEncRef:=GVL_M2L0_Constants.nYUP_ENC_REF,
               nYdwnEncRef:=GVL_M2L0_Constants.nYDWN_ENC_REF,
               nXupEncRef:=GVL_M2L0_Constants.nXUP_ENC_REF,
               nXdwnEncRef:=GVL_M2L0_Constants.nXDWN_ENC_REF,
			   bExecuteCoupleY:=M2L0.bExecuteCoupleY,
               bExecuteCoupleX:=M2L0.bExecuteCoupleX,
			   bExecuteDecoupleY:=M2L0.bExecuteDecoupleY,
               bExecuteDecoupleX:=M2L0.bExecuteDecoupleX,
               bGantryAlreadyCoupledY=>M2L0.bGantryAlreadyCoupledY,
               bGantryAlreadyCoupledX=>M2L0.bGantryAlreadyCoupledX,
               nCurrGantryY=>M2L0.nCurrGantryY,
               nCurrGantryX=>M2L0.nCurrGantryX);
fbBenderM2L0(stBender:=M12,
	         bSTOEnable1:=M2L0.fbRunHOMS.bSTOEnable1,
		     bSTOEnable2:=M2L0.fbRunHOMS.bSTOEnable2);

// Convert nCurrGantry to um (smaller number) to read out in epics
M2L0.fCurrGantryY_um := LINT_TO_REAL(M2L0.nCurrGantryY) / 1000;
M2L0.fCurrGantryX_um := LINT_TO_REAL(M2L0.nCurrGantryX) / 1000;

// FB_MotionStage's for non-piezo axes
fbMotionStage_m7(stMotionStage:=M7);
fbMotionStage_m8(stMotionStage:=M8);
fbMotionStage_m9(stMotionStage:=M9);
fbMotionStage_m10(stMotionStage:=M10);
fbMotionStage_m12(stMotionStage:=M12);

// Calculate RMS Error:
fbYRMSErrorM2L0(stMotionStage:=M7,
	            fMaxRMSError=>fMaxYRMSErrorM2L0,
				fMinRMSError=>fMinYRMSErrorM2L0);

fbXRMSErrorM2L0(stMotionStage:=M9,
	            fMaxRMSError=>fMaxXRMSErrorM2L0,
				fMinRMSError=>fMinXRMSErrorM2L0);

fbPitchRMSErrorM2L0(stMotionStage:=M11,
	                fMaxRMSError=>fMaxPitchRMSErrorM2L0,
					fMinRMSError=>fMinPitchRMSErrorM2L0);

fbBenderRMSErrorM2L0(stMotionStage:=M12,
	                 fMaxRMSError=>fMaxBenderRMSErrorM2L0,
				     fMinRMSError=>fMinBenderRMSErrorM2L0);

// Pitch Control
fbM2L0PitchControl(Pitch:=GVL_M2L0.M2L0_Pitch,
				   Stepper:=M11,
				   lrCurrentSetpoint:=M11.fPosition,
                   q_bDone=>bM2L0PitchDone,
                   q_bBusy=>bM2L0PitchBusy);
// When STO hit, need to reset SP
IF NOT M11.bHardwareEnable THEN
	M11.fPosition := M11.stAxisStatus.fActPosition;
END_IF

fbECATDiag();
fbLogHandler();

END_PROGRAM

// ---- POUs/Serial Comm/P_Serial_Com.TcPOU
PROGRAM P_Serial_Com
VAR
	fbSerialLineControl_EL6001_M1L0: SerialLineControl; // M1L0 Serial Comm Function Block
	fbSerialLineControl_EL6001_M2L0: SerialLineControl; // M2L0 Serial Comm Function Block
END_VAR

// These are the global IOs...don't forget to copy your data into them

(* EL6001 Serial port 0 com function *)
fbSerialLineControl_EL6001_M1L0(Mode:= SERIALLINEMODE_EL6_22B,
						        pComIn:= ADR(Serial_stComIn_M1L0),
						   	    pComOut:=ADR(Serial_stComOut_M1L0),
						        SizeComIn:= SIZEOF(Serial_stComIn_M1L0),
						        TxBuffer:= Serial_TXBuffer_M1L0,
						        RxBuffer:= Serial_RXBuffer_M1L0,
						        Error=>,
						        ErrorID=>);

fbSerialLineControl_EL6001_M2L0(Mode:= SERIALLINEMODE_EL6_22B,
						        pComIn:= ADR(Serial_stComIn_M2L0),
						   	    pComOut:=ADR(Serial_stComOut_M2L0),
						        SizeComIn:= SIZEOF(Serial_stComIn_M2L0),
						        TxBuffer:= Serial_TXBuffer_M2L0,
						        RxBuffer:= Serial_RXBuffer_M2L0,
						        Error=>,
						        ErrorID=>);

END_PROGRAM

// ---- POUs/Serial Comm/PiezoSerial.TcPOU
PROGRAM PiezoSerial
VAR
	//PI Serial
	fbE621SerialDriver_M1L0 : FB_PI_E621_SerialDriver;
	rtInitParams_M1L0	:	R_TRIG;
	tonTimeoutRst_M1L0	: TON := (PT:=T#2S); //For timeout reset
	
	fbE621SerialDriver_M2L0 : FB_PI_E621_SerialDriver;
	rtInitParams_M2L0	:	R_TRIG;
	tonTimeoutRst_M2L0	: TON := (PT:=T#2S); //For timeout reset
END_VAR

//Piezo E-621
///////////////////////
fbE621SerialDriver_M1L0.i_xExecute := TRUE;
fbE621SerialDriver_M1L0.i_xExecute R= fbE621SerialDriver_M1L0.q_xDone;
fbE621SerialDriver_M1L0(iq_stPiezoAxis:= GVL_M1L0.M1L0_Pitch.Piezo,
		                iq_stSerialRXBuffer:= Serial_RXBuffer_M1L0,
		                iq_stSerialTXBuffer:= Serial_TXBuffer_M1L0);

fbE621SerialDriver_M2L0.i_xExecute := TRUE;
fbE621SerialDriver_M2L0.i_xExecute R= fbE621SerialDriver_M2L0.q_xDone;
fbE621SerialDriver_M2L0(iq_stPiezoAxis:= M2L0_Pitch.Piezo,
		                iq_stSerialRXBuffer:= Serial_RXBuffer_M2L0,
		                iq_stSerialTXBuffer:= Serial_TXBuffer_M2L0);

END_PROGRAM

// ---- GlobalTextList.TcGTLO
TEXTLIST GlobalTextList
  265 = '%f'
  639 = '%X'
  631 = '+'
  625 = '-'
  635 = '0 = Default Acceleration'
  637 = '0 = Default Deceleration'
  634 = 'Acceleration: %f'
  503 = 'Already Coupled: %f'
  629 = 'Clear'
  623 = 'Control'
  862 = 'Couple Motors'
  876 = 'Couple Status: 0 = Decoupled, 1 = Coupled'
  504 = 'Couple Status: TRUE if coupled'
  220 = 'Current Gantry Difference (Axilon): %f'
  861 = 'Current Gantry Difference in um'
  860 = 'Current Gantry Difference: %f'
  266 = 'Current Position'
  636 = 'Deceleration: %f'
  871 = 'Decouple Motors'
  873 = 'Disable'
  874 = 'Enable'
  869 = 'Enable Mode: %f'
  875 = 'Enable Status: 0 = Enabled, 2 = Disabled'
  219 = 'Ensure motors are coupled before attempting motion!'
  640 = 'Error Code'
  638 = 'Error:'
  627 = 'GO'
  628 = 'GO to set position'
  267 = 'High Limit Hit Indicator'
  264 = 'Low Limit Hit Indicator'
  622 = 'Moving:'
  866 = 'Pitch - MASTER'
  863 = 'Press To Couple Motors'
  872 = 'Press To Decouple Motors for independent control'
  624 = 'Set Position'
  632 = 'Settings'
  263 = 'Status'
  626 = 'Step Size'
  630 = 'STOP'
  867 = 'Units: um'
  868 = 'Units: urad'
  633 = 'Velocity: %f'
  870 = 'Write 0 to Enable, 2 to Disable'
  865 = 'Xdwn - SLAVE'
  864 = 'Xup - MASTER'
  501 = 'Yleft - MASTER'
  502 = 'Yright - SLAVE'
END_TEXTLIST
